Universal Robots PolyScope program: g01_home.urp

Program g01_home_1 (installation=default directory=/programs createdIn=5.9.1.1031110 lastSavedIn=5.9.1.1031110 robotSerialNumber=20195501059)
Calibrated DH parameters: a=[0.000146, -0.418764, -0.053981, 0.000058, -0.000023, 0]; d=[0.162545, 37.319448, -206.067439, 168.881546, 0.09955, 0.099464]; alpha=[1.57004, -0.001979, 0.002304, 1.570607, -1.57066, 0]; deltaTheta=[0, -0.174616, -1.258233, 1.432844, -0.000001, 0]
Robot Program (runOnlyOnce=true)
  MoveJ speed 60 deg/s, acceleration 80 deg/s^2 (useActiveTCP=true) feature=Base
    Waypoint Waypoint (Variable): variable(featureName=g01_home)
  Script file /programs/g01_wrap.script
    | q = get_joint_positions()
    | q[5] = d2r(-350)
    | movej(q)
